PROGRAM MAIN
VAR

	fbMyPizzaOven:FB_PIZZA_OVEN; //oven 1
	fbMyPizzaOven2:FB_PIZZA_OVEN; //oven 2
	btn_PutAPizza:BOOL;
	btn_PackageThePizza:BOOL;
	bReset:BOOL;
	
	btn_PutAPizzaT:R_TRIG;
	btn_PackageThePizzaT:R_TRIG;
	bResetT:R_TRIG;
END_VAR

btn_PutAPizzaT(CLK:=main.btn_PutAPizza);
btn_PackageThePizzaT(CLK:=main.btn_PackageThePizza);
bResetT(CLK:=main.bReset);

fbMyPizzaOven(
	bReset:=main.bResetT.Q,
	btn_PutAPizza:=main.btn_PutAPizzaT.Q,
	btn_PackageThePizza:=main.btn_PackageThePizzaT.Q
);

fbMyPizzaOven2(
	bReset:=main.bResetT.Q,
	btn_PutAPizza:=main.btn_PutAPizzaT.Q,
	btn_PackageThePizza:=main.btn_PackageThePizzaT.Q
);

END_PROGRAM

(* stored: Version 1.1.0.1, ProductVersion 3.1.4024.3
   POU MAIN: Id {32680e72-6e98-4f5f-aa63-a3b3583f82e0}, SpecialFunc None *)
